FUNCTION_BLOCK FB_RequestChanges EXTENDS FB_IOSensor_NO IMPLEMENTS ITF_RequestChanges
VAR

END_VAR

METHOD Testing : BOOL
VAR_INPUT
END_VAR
END_METHOD

END_FUNCTION_BLOCK

(* stored: Version 1.1.0.1
   POU FB_RequestChanges: Id {ded774fa-c338-0451-01c3-5253c5ecd714}, SpecialFunc None
   Method Testing: Id {953cfe74-553d-04f4-17d9-910892e7451d} *)
